TYPE ST_APIBetweenPLC :
STRUCT
	_word: WORD;
	_int:INT;
	_Byte:BYTE;
	_String:STRING;
	_Bool:BOOL;
END_STRUCT
END_TYPE

(* stored: Version 1.1.0.1, ProductVersion 3.1.4020.12
   DUT ST_APIBetweenPLC: Id {ddd51da1-bd85-4c47-bc4e-3bc966dc0a24} *)
